TYPE (* A Structure with 16 Bits *)
  (* Version 1.0, 2024-02-21, franz *)
  st16b : STRUCT
    b00 : BOOL; (* BIT 00 *)
    b01 : BOOL; (* BIT 01 *)
    b02 : BOOL; (* BIT 02 *)
    b03 : BOOL; (* BIT 03 *)
    b04 : BOOL; (* BIT 04 *)
    b05 : BOOL; (* BIT 05 *)
    b06 : BOOL; (* BIT 06 *)
    b07 : BOOL; (* BIT 07 *)
    b08 : BOOL; (* BIT 08 *)
    b09 : BOOL; (* BIT 09 *)
    b10 : BOOL; (* BIT 10 *)
    b11 : BOOL; (* BIT 11 *)
    b12 : BOOL; (* BIT 12 *)
    b13 : BOOL; (* BIT 13 *)
    b14 : BOOL; (* BIT 14 *)
    b15 : BOOL; (* BIT 15 *)
  END_STRUCT;
END_TYPE
